SUBAPPLICATION Verteiler (* Subapplication Type *)
  (* Standard: 61499-2 *)
  (* Version 1.0, 2023-01-29, Franz *)
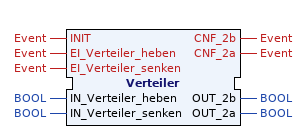
  EVENT_INPUT
    INIT;
    EI_Verteiler_heben;
    EI_Verteiler_senken;
  END_EVENT
  EVENT_OUTPUT
    CNF_2b;
    CNF_2a;
  END_EVENT
  VAR_INPUT
    IN_Verteiler_heben : BOOL;
    IN_Verteiler_senken : BOOL;
  END_VAR
  VAR_OUTPUT
    OUT_2b : BOOL;
    OUT_2a : BOOL;
  END_VAR
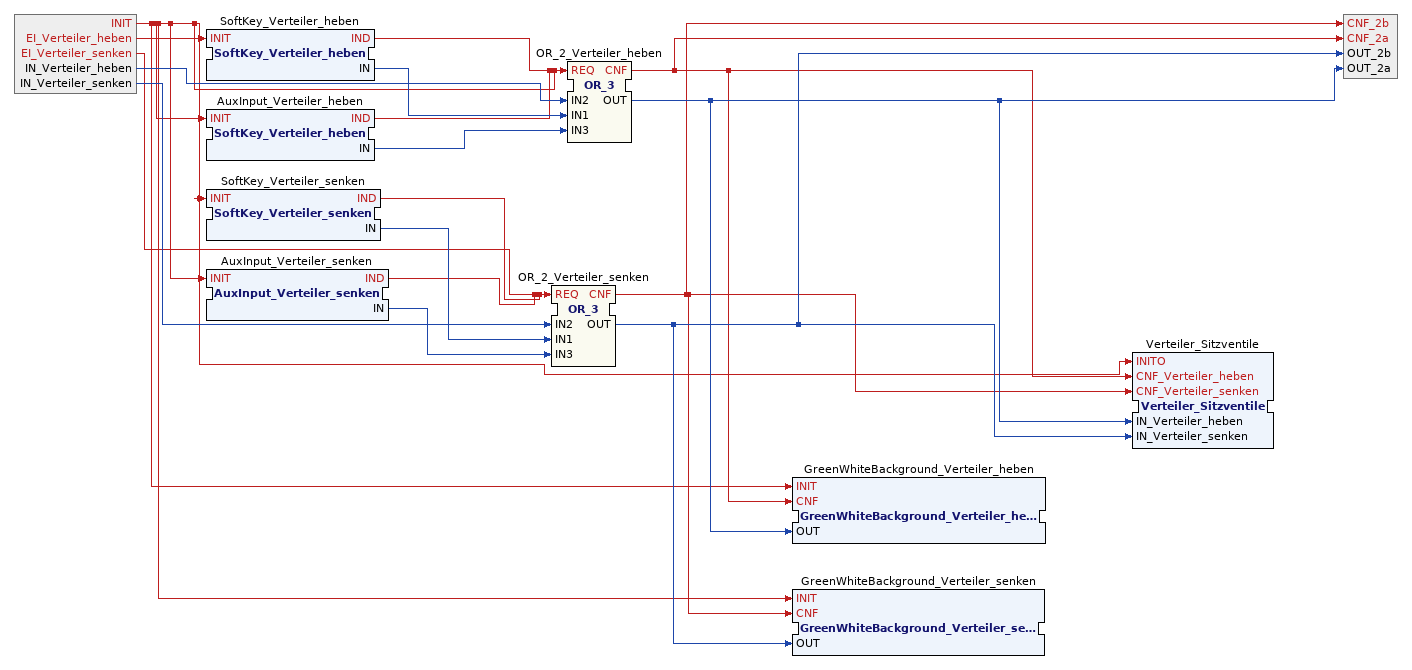
  FBS
    OR_2_Verteiler_heben : OR_3;
    OR_2_Verteiler_senken : OR_3;
  END_FBS
  SUBAPPS
    GreenWhiteBackground_Verteiler_heben : GreenWhiteBackground_Verteiler_heben;
    GreenWhiteBackground_Verteiler_senken : GreenWhiteBackground_Verteiler_senken;
    Verteiler_Sitzventile : Verteiler_Sitzventile;
    SoftKey_Verteiler_heben : SoftKey_Verteiler_heben;
    SoftKey_Verteiler_senken : SoftKey_Verteiler_senken;
    AuxInput_Verteiler_heben : SoftKey_Verteiler_heben;
    AuxInput_Verteiler_senken : AuxInput_Verteiler_senken;
  END_SUBAPPS
  EVENT_CONNECTIONS
    INIT TO GreenWhiteBackground_Verteiler_heben.INIT;
    INIT TO GreenWhiteBackground_Verteiler_senken.INIT;
    INIT TO Verteiler_Sitzventile.INITO;
    EI_Verteiler_heben TO OR_2_Verteiler_heben.REQ;
    OR_2_Verteiler_heben.CNF TO CNF_2a;
    OR_2_Verteiler_heben.CNF TO GreenWhiteBackground_Verteiler_heben.CNF;
    OR_2_Verteiler_heben.CNF TO Verteiler_Sitzventile.CNF_Verteiler_heben;
    EI_Verteiler_senken TO OR_2_Verteiler_senken.REQ;
    OR_2_Verteiler_senken.CNF TO CNF_2b;
    OR_2_Verteiler_senken.CNF TO GreenWhiteBackground_Verteiler_senken.CNF;
    OR_2_Verteiler_senken.CNF TO Verteiler_Sitzventile.CNF_Verteiler_senken;
    INIT TO SoftKey_Verteiler_heben.INIT;
    SoftKey_Verteiler_heben.IND TO OR_2_Verteiler_heben.REQ;
    INIT TO SoftKey_Verteiler_senken.INIT;
    SoftKey_Verteiler_senken.IND TO OR_2_Verteiler_senken.REQ;
    INIT TO AuxInput_Verteiler_heben.INIT;
    AuxInput_Verteiler_heben.IND TO OR_2_Verteiler_heben.REQ;
    INIT TO AuxInput_Verteiler_senken.INIT;
    AuxInput_Verteiler_senken.IND TO OR_2_Verteiler_senken.REQ;
  END_CONNECTIONS
  DATA_CONNECTIONS
    IN_Verteiler_heben TO OR_2_Verteiler_heben.IN2;
    OR_2_Verteiler_heben.OUT TO OUT_2a;
    OR_2_Verteiler_heben.OUT TO GreenWhiteBackground_Verteiler_heben.OUT;
    OR_2_Verteiler_heben.OUT TO Verteiler_Sitzventile.IN_Verteiler_heben;
    IN_Verteiler_senken TO OR_2_Verteiler_senken.IN2;
    OR_2_Verteiler_senken.OUT TO OUT_2b;
    OR_2_Verteiler_senken.OUT TO GreenWhiteBackground_Verteiler_senken.OUT;
    OR_2_Verteiler_senken.OUT TO Verteiler_Sitzventile.IN_Verteiler_senken;
    SoftKey_Verteiler_heben.IN TO OR_2_Verteiler_heben.IN1;
    SoftKey_Verteiler_senken.IN TO OR_2_Verteiler_senken.IN1;
    AuxInput_Verteiler_heben.IN TO OR_2_Verteiler_heben.IN3;
    AuxInput_Verteiler_senken.IN TO OR_2_Verteiler_senken.IN3;
  END_CONNECTIONS
END_SUBAPPLICATION
